PROGRAM TimeControl
VAR
END_VAR

// NETWORK 1

END_PROGRAM

(* stored: Version 1.1.0.1, ProductVersion 3.1.4024.12
   POU TimeControl: Id {50f369aa-c81b-463a-bb19-632e394a17ea}, SpecialFunc None *)
